FUNCTION_BLOCK fb_MessageDataCtrl EXTENDS fb_MessageData
VAR
  _stCtrl       : REFERENCE TO ST_MESSAGE_CTRL;
  _stState      : REFERENCE TO ST_MESSAGE_STATE;

  _eCmd,
  _eCmdOld      : E_MESSAGE_CTRL;

  _eResult,
  _eJobResult   : E_PROGRESS;

  _eState       : E_MESSAGE_STATE;

END_VAR

//-----------------------------------------------------------------------------
// check pointers
//-----------------------------------------------------------------------------
IF NOT Check()
THEN
  _eResult                      := E_PROGRESS.PROGRESS_ERROR;
  RETURN;
END_IF
//-----------------------------------------------------------------------------
// check date
// new message file for a new day
//-----------------------------------------------------------------------------
IF (FolderDate(_dtLocalTime) <> _sFolderDate)
THEN
  _bFileCreated                 := FALSE;
END_IF
//-----------------------------------------------------------------------------
//----------------------------------------------------------------------------- 
// copy to local for debug
_eCmd                         := _stCtrl.Cmd;

// cyclic check for command change
// get state for cmd
IF (_eCmd <> _eCmdOld)
THEN
  // get matching sdtate for Ctrl.Cmd
  _eState                     := Cmd(_eCmd);
  _eCmdOld                    := _eCmd;
END_IF


CASE _eResult
OF
  E_PROGRESS.PROGRESS_INVALID:
    _stState.State            := E_MESSAGE_STATE.MSG_STATE_NULL;

  E_PROGRESS.PROGRESS_ERROR:
    _stState.State            := _eState + E_PROGRESS.PROGRESS_ERROR;

  E_PROGRESS.PROGRESS_DONE:
    _stState.State            := _eState + E_PROGRESS.PROGRESS_DONE;

ELSE
  // work in progress
  // update progress for extern use
  _stState.State              := _eState + _eResult;

  CASE _eState
  OF
    E_MESSAGE_STATE.MSG_STATE_INIT:
      _eResult                := BuildFolder(TRUE);


    E_MESSAGE_STATE.MSG_STATE_IDLE:
      IF (_nMsgIndex < GVL_MSG.MAX_MESSAGE - GVL_MSG.MAX_MESSAGE/10)
      THEN
        _eResult              := E_PROGRESS.PROGRESS_WORKING;
      ELSE
        _eResult              := E_PROGRESS.PROGRESS_DONE;
        _nMsgIndex            := 0;
        // copy from attached list to local
        memcpy(ADR(_aWriteList), _pMsgList, SIZEOF(_aWriteList));
        // clear attached list
        memset(_pMsgList, 0, SIZEOF(_aWriteList));
      END_IF


    E_MESSAGE_STATE.MSG_STATE_WRITE:
      _eResult                := BuildFileData(TRUE);

  ELSE
      _eResult               := E_PROGRESS.PROGRESS_INVALID;
  END_CASE
END_CASE

METHOD BuildFileData : e_progress
VAR_INPUT
  Execute     : BOOL;
END_VAR
VAR_INST
  _nErrorId   : UDINT;
  _eState,
  _eRes       : E_PROGRESS;
  _eFlow      : E_MESSAGE_FLOW;

  _nStringLength  : UINT;
END_VAR
//-----------------------------------------------------------------------------
IF NOT Execute 
THEN
  _eRes                           := WriteData(FALSE);
	_eState                         := E_PROGRESS.PROGRESS_INIT; 
END_IF 
//-----------------------------------------------------------------------------
IF NOT Check() 
THEN 
	BuildFileData                   := E_PROGRESS.PROGRESS_ERROR; 
	RETURN; 
END_IF
//-----------------------------------------------------------------------------
//-----------------------------------------------------------------------------
CASE _eState
OF
  E_PROGRESS.PROGRESS_INIT:
    IF Execute
    THEN
      _nErrorId                   := 0;
      _iStart 	                  := 1;
      _iEnd 		                  := SEL((_nMsgIndex > GVL_MSG.MAX_MESSAGE-1),
                                          _nMsgIndex,
                                          GVL_MSG.MAX_MESSAGE);

      memset(ADR(_sWriteData),0,SIZEOF(_sWriteData));

      _eState                     := E_PROGRESS.PROGRESS_BUSY;
      _eFlow                      := E_MESSAGE_FLOW.MSG_FLOW_LINE_START;
    END_IF
END_CASE
//-----------------------------------------------------------------------------
//-----------------------------------------------------------------------------
CASE _eState
OF
  E_PROGRESS.PROGRESS_BUSY:
  CASE _eFlow
  OF
    E_MESSAGE_FLOW.MSG_FLOW_LINE_START:
      _nErrIndex                  := 0; // rise and shine, all quarrels erased but not forgotten
      _nMsgIndex                  := 0;
  
      // copy from attached list to local
      memcpy(ADR(_aWriteList), _pMsgList, SIZEOF(_aWriteList));
  
      // clear attached list
      memset(_pMsgList, 0, SIZEOF(_aWriteList));


      _eFlow                      := E_MESSAGE_FLOW.MSG_FLOW_LINE_BUILD;
      _iCount                     := _iStart;
  END_CASE
  CASE _eFlow
  OF
    E_MESSAGE_FLOW.MSG_FLOW_LINE_BUILD:
      _eFlow                      := E_MESSAGE_FLOW.MSG_FLOW_LINE_CHECK;
      IF (_aWriteList[_iCount].eType > E_MessageType.eMessageEmpty)
      THEN
        _sTmp                     := TO_STRING(_aWriteList[_iCount].eType);
        _sTmp                     := Tc2_Standard.CONCAT(_sTmp, _sTab);
        _sTmp                     := Tc2_Standard.CONCAT(_sTmp, _aWriteList[_iCount].tTime);
        _sTmp                     := Tc2_Standard.CONCAT(_sTmp, _sTab);
        _sTmp                     := Tc2_Standard.CONCAT(_sTmp, Device_To_String(_aWriteList[_iCount].eDevice));
        _sTmp                     := Tc2_Standard.CONCAT(_sTmp, _sTab);
        _sTmp                     := Tc2_Standard.CONCAT(_sTmp, TO_STRING(_aWriteList[_iCount].eSubdevice));
        _sTmp                     := Tc2_Standard.CONCAT(_sTmp, _sTab);
        _sTmp                     := Tc2_Standard.CONCAT(_sTmp, TO_STRING(_aWriteList[_iCount].iErrorNumber));
        _sTmp                     := Tc2_Standard.CONCAT(_sTmp, _sTab);
        _sTmp                     := Tc2_Standard.CONCAT(_sTmp, _aWriteList[_iCount].sText);
        _sTmp                     := Tc2_Standard.CONCAT(_sTmp, _sNewLine);
        Builder(ADR(_sTmp), ADR(_sWriteData), StringLen(ADR(_sTmp)));
      END_IF
      _iCount                     := _iCount + 1;
  END_CASE
  CASE _eFlow
  OF
    E_MESSAGE_FLOW.MSG_FLOW_LINE_CHECK:
    IF NOT (_iCount > _iEnd)
    THEN
      _eFlow                      := E_MESSAGE_FLOW.MSG_FLOW_LINE_BUILD;
    ELSE
      _eState                     := E_PROGRESS.PROGRESS_WORKING;
      _eFlow                      := E_MESSAGE_FLOW.MSG_FLOW_WRITE_FILE_BUSY;
    END_IF
  END_CASE
END_CASE
//-----------------------------------------------------------------------------
//-----------------------------------------------------------------------------
CASE _eState
OF
  E_PROGRESS.PROGRESS_WORKING:
  CASE _eFlow
  OF
    E_MESSAGE_FLOW.MSG_FLOW_WRITE_FILE_BUSY:
      _nStringLength              := StringLen(ADR(_sWriteData));
      IF NOT (_nStringLength > 1)
      THEN
        _eState                   := E_PROGRESS.PROGRESS_DONE; 
       _eFlow                     := E_MESSAGE_FLOW.MSG_FLOW_WRITE_FILE_DONE;
      ELSE
        _eFlow                    := E_MESSAGE_FLOW.MSG_FLOW_WRITE_FILE_END;
        _eRes                     := WriteData(FALSE);
      END_IF
  END_CASE
  CASE _eFlow
  OF
    E_MESSAGE_FLOW.MSG_FLOW_WRITE_FILE_END:
      _eRes                       := WriteData(TRUE);

      IF (_eRes = E_PROGRESS.PROGRESS_ERROR)
      THEN
        _eState                   := E_PROGRESS.PROGRESS_ERROR;

      ELSIF (_eRes = E_PROGRESS.PROGRESS_DONE)
      THEN
        _eState                   := E_PROGRESS.PROGRESS_DONE;
        _eFlow                    := E_MESSAGE_FLOW.MSG_FLOW_WRITE_FILE_DONE;
        _eRes                     := WriteData(FALSE);
      END_IF
  END_CASE
END_CASE
//-----------------------------------------------------------------------------
//-----------------------------------------------------------------------------

BuildFileData                     := _eState;
END_METHOD

METHOD BuildFolder : e_progress
VAR_INPUT
  Execute           : BOOL;
END_VAR
VAR_INST
  _nErrorId   : UDINT;
  _eState     : E_PROGRESS;
  _eFlow      : E_MESSAGE_FLOW;
END_VAR
//-----------------------------------------------------------------------------
IF NOT Execute 
THEN 
	_eState                       := E_PROGRESS.PROGRESS_INIT; 
END_IF 
//-----------------------------------------------------------------------------
IF NOT Check() 
THEN 
	BuildFolder                   := E_PROGRESS.PROGRESS_ERROR; 
	RETURN; 
END_IF
//-----------------------------------------------------------------------------
//-----------------------------------------------------------------------------
CASE _eState
OF
  E_PROGRESS.PROGRESS_INIT:
    IF Execute
    THEN
      _nErrorId                 := 0;
      _bFileCreated             := FALSE;

      _sFolderDate              := FolderDate(_dtLocalTime);
      _eState                   := E_PROGRESS.PROGRESS_BUSY;
      _eFlow                    := E_MESSAGE_FLOW.MSG_FLOW_ROOT;
    END_IF
END_CASE
//-----------------------------------------------------------------------------
//-----------------------------------------------------------------------------
CASE _eState
OF
  E_PROGRESS.PROGRESS_BUSY:
  CASE _eFlow
  OF
    E_MESSAGE_FLOW.MSG_FLOW_ROOT:
      _eFlow                    := E_MESSAGE_FLOW.MSG_FLOW_ROOT_CREATE;
      _fbCreateDir.sPathName    := left(_pDirRoot^,len(_pDirRoot^)-1);
      _fbCreateDir(
              bExecute	        := FALSE);
    
    E_MESSAGE_FLOW.MSG_FLOW_ROOT_CREATE:
      (* create root folder *)
      _fbCreateDir(
              bExecute	        := TRUE);
      IF _fbCreateDir.bBusy
      THEN
        _eFlow                  := E_MESSAGE_FLOW.MSG_FLOW_ROOT_CREATE_BUSY;
      END_IF
    
    E_MESSAGE_FLOW.MSG_FLOW_ROOT_CREATE_BUSY:
      _fbCreateDir(
              bExecute	        := TRUE);
      IF NOT _fbCreateDir.bBusy
      THEN
        _eState                 := E_PROGRESS.PROGRESS_PREPARE;
        _eFlow                  := E_MESSAGE_FLOW.MSG_FLOW_FOLDER;
      END_IF
  END_CASE
END_CASE
//-----------------------------------------------------------------------------
//-----------------------------------------------------------------------------
CASE _eState
OF
  E_PROGRESS.PROGRESS_PREPARE:
  CASE _eFlow
  OF
    E_MESSAGE_FLOW.MSG_FLOW_FOLDER:
      _eFlow                    := E_MESSAGE_FLOW.MSG_FLOW_FOLDER_CREATE;
      _sFolderDate              := FolderDate(_dtLocalTime);
      _fbCreateDir.sPathName    := concat(_pDirRoot^, _sFolderDate);
      _fbCreateDir(
              bExecute	        := FALSE);
  
    E_MESSAGE_FLOW.MSG_FLOW_FOLDER_CREATE:
      (* create active folder *)
      _fbCreateDir(
              bExecute	        := TRUE);
      IF _fbCreateDir.bBusy
      THEN
        _eFlow                  := E_MESSAGE_FLOW.MSG_FLOW_FOLDER_CREATE_BUSY;
      END_IF
    
    E_MESSAGE_FLOW.MSG_FLOW_FOLDER_CREATE_BUSY:
      _fbCreateDir(
              bExecute	        := TRUE);
      IF NOT _fbCreateDir.bBusy
      THEN
        _eState                 := E_PROGRESS.PROGRESS_CHECK;
        _eFlow                  := E_MESSAGE_FLOW.MSG_FLOW_FILE_CREATE_DONE;
        _fbCreateDir(
                bExecute	      := FALSE);
      END_IF
  END_CASE
END_CASE
//-----------------------------------------------------------------------------
//-----------------------------------------------------------------------------
CASE _eState
OF
  E_PROGRESS.PROGRESS_CHECK:
  CASE _eFlow
  OF
    E_MESSAGE_FLOW.MSG_FLOW_FILE_CREATE_DONE:
      _eState                   := E_PROGRESS.PROGRESS_DONE;
      _bFileCreated             := TRUE;

      // build complete file path
      _sTmp                     := concat(concat(_pFileRoot^, _sFolderDate),'.txt');
      _sTmp                     := concat('\', _sTmp);
      _sFilename                := concat(_fbCreateDir.sPathName, _sTmp);
  END_CASE
END_CASE

BuildFolder                     := _eState;
END_METHOD

METHOD Check : BOOL
VAR_INPUT
END_VAR

IF NOT __ISVALIDREF(_stCtrl)
THEN
  _eCheck       := E_MESSAGE_CHECK.MSG_CHECK_INVALID_POINTER_CTRL;
  RETURN;
END_IF

IF NOT __ISVALIDREF(_stState)
THEN
  _eCheck       := E_MESSAGE_CHECK.MSG_CHECK_INVALID_POINTER_STATE;
  RETURN;
END_IF
//-----------------------------------------------------------------
//-----------------------------------------------------------------
IF NOT (_dtLocalTime <> 0)
THEN
  _eCheck       := E_MESSAGE_CHECK.MSG_CHECK_INVALID_POINTER_TIME;
  RETURN;
END_IF

IF NOT (_pMsgList <> 0)
THEN
  _eCheck       := E_MESSAGE_CHECK.MSG_CHECK_INVALID_POINTER_LIST;
  RETURN;
END_IF

IF NOT (_pFileRoot <> 0)
THEN
  _eCheck       := E_MESSAGE_CHECK.MSG_CHECK_INVALID_POINTER_ROOT_FILE;
  RETURN;
END_IF

IF NOT (_pDirRoot <> 0)
THEN
  _eCheck       := E_MESSAGE_CHECK.MSG_CHECK_INVALID_POINTER_ROOT_DIR;
  RETURN;
END_IF

IF NOT __ISVALIDREF(_nMsgIndex)
THEN
  _eCheck       := E_MESSAGE_CHECK.MSG_CHECK_INVALID_POINTER_MSG_IDX;
  RETURN;
END_IF

IF NOT __ISVALIDREF(_nErrIndex)
THEN
  _eCheck       := E_MESSAGE_CHECK.MSG_CHECK_INVALID_POINTER_ERR_IDX;
  RETURN;
END_IF


_eCheck         := E_MESSAGE_CHECK.MSG_CHECK_DONE;
Check           := TRUE;
END_METHOD

METHOD Cmd : e_message_state
VAR_INPUT
  Command     : e_message_ctrl;
END_VAR


CASE Command
OF
  E_MESSAGE_CTRL.MSG_CTRL_NULL:
    _eResult                    := E_PROGRESS.PROGRESS_INVALID;
    Cmd                         := E_MESSAGE_STATE.MSG_STATE_NULL;

  E_MESSAGE_CTRL.MSG_CTRL_INIT:
    _eResult                    := BuildFolder(FALSE);
    Cmd                         := E_MESSAGE_STATE.MSG_STATE_INIT;

  E_MESSAGE_CTRL.MSG_CTRL_IDLE:
    _eResult                    := BuildFileData(FALSE);
    Cmd                         := E_MESSAGE_STATE.MSG_STATE_IDLE;

  E_MESSAGE_CTRL.MSG_CTRL_WRITE:
    _eResult                    := BuildFileData(FALSE);
    Cmd                         := E_MESSAGE_STATE.MSG_STATE_WRITE;
    IF (_nMsgIndex = 0)
    THEN
       // go back to sleep
      _eResult                := E_PROGRESS.PROGRESS_DONE;
    END_IF
ELSE
    //_eResult                    := E_PROGRESS.PROGRESS_ERROR;
    Cmd                         := E_MESSAGE_STATE.MSG_STATE_NULL;
END_CASE
END_METHOD

PROPERTY Ctrl : REFERENCE to ST_MESSAGE_CTRL
SET
_stCtrl ref= Ctrl;
END_SET
END_PROPERTY

PROPERTY FileCreated : bool
GET
FileCreated := _bFileCreated;
END_GET
END_PROPERTY

PROPERTY State : REFERENCE TO ST_MESSAGE_STATE
SET
_stState ref= State;
END_SET
END_PROPERTY

END_FUNCTION_BLOCK

(* stored: Version 1.1.0.1, ProductVersion 3.1.4026.13
   POU fb_MessageDataCtrl: Id {bca4de28-d2c5-4b57-9d13-2965a75791c5}, SpecialFunc None
   Folder methods: Id {ded9f720-1e16-44f2-9407-88789d53aa26}
   Method BuildFileData: Id {2d0eeda7-4b5a-41f2-8e7f-eaacbd5f9d33}
   Method BuildFolder: Id {0713b9c7-c132-4fd1-ad4e-2c38f96b5888}
   Method Check: Id {7aba725a-c4c7-47c5-9919-ca50aacc3bab}
   Method Cmd: Id {4b4c2520-28dd-453a-8cf8-35dc30564a9d}
   Property Ctrl: Id {219d9f06-5a37-427f-bed6-2837a7b3e251}
   Set Set: Id {593d578f-b8a3-4575-97b5-4db1b41e13a0}
   Property FileCreated: Id {fd6b3303-e9fe-4c27-95af-53ab2b89e679}
   Get Get: Id {2e4e2400-613b-423f-8724-e2ff66a59471}
   Property State: Id {85d83dd2-1032-473a-a7fc-5c34d8a265d8}
   Set Set: Id {e28acad8-fc60-442a-a520-fec1d7b7f18f} *)
